// v2 moved ConflictTime to ST_AirPressureStationCfg: it varies per
// deployment, not per model, and §3.8a places such a value in station
// configuration. This monitor has no model data of its own, so what remains
// is the versioned shell the §3.12 contract asks every module to carry.
TYPE ST_AirPressureParCfg :
STRUCT
    SchemaVersion : UINT := 2;       // §3.8: MUST remain first
END_STRUCT
END_TYPE

(* stored: Version 1.1.0.1, ProductVersion 3.1.4024.12
   DUT ST_AirPressureParCfg: Id {bad76f9a-9f1b-4d9a-9479-1b5286b636b7} *)
